{attribute 'linkalways'} 
{attribute 'no_explicit_call' := 'This FB is a CLASS and must be accessed using methods or properties'}
{attribute 'enable_dynamic_creation'}
FUNCTION_BLOCK Node_F_VN_AppendToContainer_TcVnVector4_UINT EXTENDS VisionNode
VAR
    aElement : _TcVnVector4_UINT;
    ipContainer : _ITcVnContainer;
    hrPrev : _HRESULT(S_OK);
	hresult : _HRESULT(S_OK);
END_VAR

METHOD PUBLIC  Clone : I_Node
VAR
	pNode : POINTER TO Node_F_VN_AppendToContainer_TcVnVector4_UINT;
END_VAR
pNode := __NEW(Node_F_VN_AppendToContainer_TcVnVector4_UINT);
Clone := pNode^;
END_METHOD

METHOD FB_init : BOOL
VAR_INPUT
	bInitRetains : BOOL; // if TRUE, the retain variables are initialized (warm start / cold start)
	bInCopyCode : BOOL;  // if TRUE, the instance afterwards gets moved into the copy code (online change)
END_VAR
AddInput('aElement', aElement);
AddInput('ipContainer', ipContainer);
AddInput('hrPrev', hrPrev);
AddOutput('ipContainer', ipContainer);
AddOutput('hresult',hresult);
END_METHOD

METHOD PROTECTED OnExecute
hresult.Value := F_VN_AppendToContainer_TcVnVector4_UINT(
    aElement := aElement.Value,
	ipContainer := ipContainer.Value,
	hrPrev:= hrPrev.Value);
END_METHOD

METHOD PUBLIC PreExecutionCheck
VAR_INPUT
	Check : I_PreExecutionChecks;
END_VAR
Check.IsTrue(ipContainer.IsValid, 'ipContainer must be a valid container');
Check.IsTrue(ipContainer.IsType(TC_GLOBAL_CONST_LIST.ContainerType_Vector_TcVnVector4_UINT), 'ipContainer contains incorrect type');
END_METHOD

END_FUNCTION_BLOCK

(* stored: Version 1.1.0.1, ProductVersion 3.1.4026.13
   POU Node_F_VN_AppendToContainer_TcVnVector4_UINT: Id {cb78c7ce-d101-4289-b7e0-6c94456c8aa7}, SpecialFunc None
   Folder Constructor: Id {2c07c5b4-09b1-4d91-bf83-d9783db55469}
   Method Clone: Id {4db206f0-19d2-46a2-9a9f-104c31abe6ca}
   Method FB_init: Id {4f8ea3fb-a0f4-4a99-9b1f-404d6c41aaa6}
   Method OnExecute: Id {048972c6-b981-4449-a55a-aa35360d831e}
   Method PreExecutionCheck: Id {d55a4d8c-b825-4420-83e9-c9f1e225d175} *)
